FUNCTION_BLOCK FB_WFSTest EXTENDS FB_TestSuite
VAR
    (* Caller-owned axis, persistent storage, and Y motor.
       In a real PRG the AxisRef would come from MAIN.Mxx. *)
    axRef    : AXIS_REF;
    fbPDS    : LCLS_Tc_DevAbs.FB_PersistentDataStorage;

    (* FB_WFS is single-axis (nActiveMotorCount := 1), so only slot 1
       holds a real motor. aiMotionStage is sized to
       MotionConstants.MAX_STATE_MOTORS to match FB_WFS.FB_Init's
       fixed-size signature; slots 2-4 default-init to a nil interface
       and are never touched. *)
    fbMotorY : FB_MotionStageNC(AxisRef := axRef, iPersistentDataStorage := fbPDS, sName := 'Y');
    aiMotionStage : ARRAY[1..MotionConstants.MAX_STATE_MOTORS] OF I_MotionStage := [fbMotorY];

    {attribute 'pytmc' := '
        pv: MMS
        astPositionState.array: 1..6
    '}
    astPositionState : ARRAY[1..MotionConstants.MAX_STATE_MOTORS]
                         OF ARRAY[1..GeneralConstants.MAX_STATES] OF ST_PositionState;

    fbFFHWO    : FB_HardwareFFOutput;
    fbArbiter  : FB_Arbiter(1);
    fbSubSysIO : FB_DummyArbIO;

    sDeviceName    : STRING := 'TST:WFS';
    sTransitionKey : STRING := 'TST:WFS-TRANSITION';

    (* Caller-owned file-reader status, bound to FB_WFS by REFERENCE
       TO. In a real PRG these point at MOTION_GVL.fbPmpsFileReader;
       here they stay FALSE so the DB read proceeds. *)
    bFileReaderBusy  : BOOL;
    bFileReaderError : BOOL;

    fbWFS : FB_WFS(
        aiMotionStage         := aiMotionStage,
        astPositionState      := astPositionState,
        fbFFHWO               := fbFFHWO,
        fbArbiter             := fbArbiter,
        sDeviceName           := sDeviceName,
        sTransitionKey        := sTransitionKey,
        bEnableBeamParams     := TRUE,
        bEnablePositionLimits := TRUE,
        bReadDBNow            := TRUE,
        bFileReaderBusy       := bFileReaderBusy,
        bFileReaderError      := bFileReaderError
    );

    (* Per-install PMPS-side state config (caller-owned). Mirrors what
       a real PRG_xxL0_WFS would declare. stDefault is the caller-owned
       baseline template that FB_CC_StatePMPSConfig's inner FB_StateSetup
       preloads from; fbWFS subsequently overrides per-state sName and
       fDelta via its own FB_CC_DeviceStateDefaults array. *)
    stDefault : ST_PositionState := (
        bMoveOk       := TRUE,
        bValid        := TRUE,
        bUseRawCounts := FALSE
    );

    afbStatePMPS : ARRAY[1..6] OF FB_CC_StatePMPSConfig[
        (stPositionState := astPositionState[1][E_WFS_States.OUT],
         stDefault       := stDefault,
         fPosition       := 10,
         sPmpsState      := 'TST:WFS-OUT'),
        (stPositionState := astPositionState[1][E_WFS_States.TARGET1],
         stDefault       := stDefault,
         fPosition       := 20,
         sPmpsState      := 'TST:WFS-TARGET1'),
        (stPositionState := astPositionState[1][E_WFS_States.TARGET2],
         stDefault       := stDefault,
         fPosition       := 30,
         sPmpsState      := 'TST:WFS-TARGET2'),
        (stPositionState := astPositionState[1][E_WFS_States.TARGET3],
         stDefault       := stDefault,
         fPosition       := 40,
         sPmpsState      := 'TST:WFS-TARGET3'),
        (stPositionState := astPositionState[1][E_WFS_States.TARGET4],
         stDefault       := stDefault,
         fPosition       := 50,
         sPmpsState      := 'TST:WFS-TARGET4'),
        (stPositionState := astPositionState[1][E_WFS_States.TARGET5],
         stDefault       := stDefault,
         fPosition       := 60,
         sPmpsState      := 'TST:WFS-TARGET5')
    ];

    bFirstScan : BOOL := TRUE;
    i          : UINT;
END_VAR

(* Fake PMPS handling. *)
fbSubSysIO(
    LA  := fbArbiter,
    FFO := fbFFHWO
);

(* Caller-side PMPS configurators write each slot once in
   FB_CC_StatePMPSConfig.CallAfterInit; no cyclic tick. *)

(* One-shot motor setup + initial caller-owned enables. Limits,
   brake/enable modes, home cmd, user/hardware enables, default
   velocity; skip NC param restore. *)
IF bFirstScan THEN
    fbMotorY.SetModeEnableLimits(
        LimBackward    := TRUE,
        LimForward     := TRUE,
        HomeEnable     := FALSE,
        BrakeMode      := E_StageBrakeMode.IF_ENABLED,
        EnableMode     := E_StageEnableMode.DURING_MOTION,
        HomeMode       := E_EpicsHomeCmd.LOW_LIMIT,
        UserEnable     := TRUE,
        HardwareEnable := TRUE
    );
    fbMotorY.SetVelocity(Velocity := 15.5);
    fbMotorY.RestoreMotionParams      := FALSE;
    fbMotorY.DoNotRestoreNcParameters := TRUE;

    bFirstScan := FALSE;
END_IF

fbPDS();
fbMotorY();
fbWFS();

TestStateMove();
TestTempFFO();

METHOD SetWFSTemp
VAR_INPUT
    iTempC : INT;
END_VAR
VAR
    ptr : POINTER TO INT;
END_VAR
ptr  := ADR(fbWFS.fbThermoCouple1.iRaw);
ptr^ := iTempC * 10;

ptr  := ADR(fbWFS.fbThermoCouple2.iRaw);
ptr^ := iTempC * 10;
END_METHOD

(*
    Smoke test for WFS state-move wiring. Walks OUT then TARGET1 and
    asserts each lands within fTolerance of the configured fPosition.
    Mirrors FB_REFTest: stageReady gate up front, NOT bMoving +
    position-tolerance check per state, 60s watchdog, on timeout
    AssertTrue(FALSE, ...) with the current step and observed
    position. Two moves is enough to exercise the FB wiring; the
    motion stack itself is covered by the
    lcls-twincat-motion-abstraction test suite.
*)
METHOD TestStateMove
VAR_INST
    tonTimer  : TON;
    nTestStep : INT := 0;
    fObserved : LREAL;
END_VAR
VAR CONSTANT
    fTolerance : LREAL := 2.0;
END_VAR
TEST('TestWFSStateMove');

tonTimer(IN := TRUE, PT := T#60s);
fObserved := fbMotorY.stMotionStatus.fActPosition;

CASE nTestStep OF
    0:
        IF fbMotorY.stMotionStatus.bStageReady
           AND NOT fbMotorY.stMotionStatus.bError THEN
            fbWFS.eEnumSet := E_WFS_States.OUT;
            nTestStep      := 1;
        END_IF
    1:
        (* OUT is configured at fPosition := 10 in afbStatePMPS[1]. *)
        IF fbWFS.eEnumGet = E_WFS_States.OUT
           AND NOT fbMotorY.stMotionStatus.bMoving
           AND ABS(fObserved - 10.0) <= fTolerance THEN
            fbWFS.eEnumSet := E_WFS_States.TARGET1;
            nTestStep      := 2;
        END_IF
    2:
        (* TARGET1 is configured at fPosition := 20 in afbStatePMPS[2]. *)
        IF fbWFS.eEnumGet = E_WFS_States.TARGET1
           AND NOT fbMotorY.stMotionStatus.bMoving
           AND ABS(fObserved - 20.0) <= fTolerance THEN
            AssertTrue(
                Condition := TRUE,
                Message   := 'TestWFSStateMove: OUT then TARGET1 reached within tolerance');
            nTestStep := 3;
        END_IF
END_CASE

IF nTestStep = 3 THEN
    TEST_FINISHED();
ELSIF tonTimer.Q THEN
    AssertTrue(
        Condition := FALSE,
        Message   := CONCAT(
            CONCAT(
                CONCAT('TestWFSStateMove: timed out at step ', TO_STRING(nTestStep)),
                CONCAT(', eEnumGet=', TO_STRING(TO_UDINT(fbWFS.eEnumGet)))),
            CONCAT(', fActPos=', TO_STRING(fObserved))));
    TEST_FINISHED();
END_IF
END_METHOD

METHOD TestTempFFO
VAR_INST
    tonTimer    : TON;
    nStep       : UINT := 0;
    bOutChecked : BOOL := FALSE;
    bInChecked  : BOOL := FALSE;
END_VAR
VAR CONSTANT
    nLastStep : UINT := 3;
END_VAR

(* Do we fault at the correct times?
   Parasitically depends on state move test. *)
TEST('TestWFSTempFFO');

(* Prepare a timeout *)
tonTimer(IN := TRUE, PT := T#10s);

CASE nStep OF
    0:
        (* Set both thermocouple temperatures to crazy high number. *)
        SetWFSTemp(100);
        nStep := nStep + 1;
    1:
        (* Wait till we see "OUT" state and one other state (OUT
           should be no fault). *)
        IF fbWFS.eEnumGet = E_WFS_States.OUT THEN
            AssertTrue(
                fbWFS.fbThermoCouple1.FFO.i_xOK,
                'TC1 faulted even in out position!'
            );
            AssertTrue(
                fbWFS.fbThermoCouple2.FFO.i_xOK,
                'TC2 faulted even in out position!'
            );
            bOutChecked := TRUE;
        ELSIF fbWFS.eEnumGet <> E_WFS_States.Unknown THEN
            AssertFalse(
                fbWFS.fbThermoCouple1.FFO.i_xOK,
                'TC1 no fault even for an in position!'
            );
            AssertFalse(
                fbWFS.fbThermoCouple2.FFO.i_xOK,
                'TC2 no fault even for an in position!'
            );
            bInChecked := TRUE;
        END_IF
        IF bOutChecked AND bInChecked THEN
            nStep := nStep + 1;
        END_IF
    2:
        (* Set both thermocouple temperatures to low again. *)
        SetWFSTemp(0);
        nStep := nStep + 1;
    3:
        AssertTrue(
            fbWFS.fbThermoCouple1.FFO.i_xOK,
            'TC1 faulted even with low temp!'
        );
        AssertTrue(
            fbWFS.fbThermoCouple2.FFO.i_xOK,
            'TC2 faulted even with low temp!'
        );
        nStep := nStep + 1;
END_CASE

IF tonTimer.Q OR nStep > nLastStep THEN
    AssertFalse(tonTimer.Q, 'Timeout in WFS temp FFO test');
    TEST_FINISHED();
END_IF
END_METHOD

END_FUNCTION_BLOCK

(* stored: Version 1.1.0.1
   POU FB_WFSTest: Id {d781df70-ea58-464c-9c90-20fbc2746e0a}, SpecialFunc None
   Method SetWFSTemp: Id {d1268d1a-3c93-46a7-bd70-abc42ffcf929}
   Method TestStateMove: Id {a0e8e497-91d8-4707-b6b1-4494ed854f9c}
   Method TestTempFFO: Id {1b4ac7c4-07b0-4d1a-97dd-2dfd68cd11c9} *)
